FUNCTION_BLOCK FB_LinkDataByte EXTENDS FB_LinkDevice
VAR	
	ControlData		AT %Q* : BYTE; //{simulation-interface}
	StatusData		AT %I* : BYTE; //{simulation-interface}	
END_VAR

SUPER^();

METHOD INTERNAL GetLinkControlData : BYTE
GetLinkControlData := ControlData;
END_METHOD

METHOD INTERNAL SetLinkStatusData : BOOL
VAR_INPUT
	nStatusData : BYTE;
END_VAR
StatusData := nStatusData;
END_METHOD

END_FUNCTION_BLOCK

(* stored: Version 1.1.0.1, ProductVersion 3.1.4024.12
   POU FB_LinkDataByte: Id {d6694e9a-755c-0867-08ff-7028877ecfeb}, SpecialFunc None
   Method GetLinkControlData: Id {4dd37bc7-9049-0901-256f-62c7bbeec0ed}
   Method SetLinkStatusData: Id {b82aec9e-0c4e-0178-1e4e-ae62bf953488} *)
